PROGRAM MAIN
VAR
END_VAR

Control_FBD();

END_PROGRAM

(* stored: Version 1.1.0.1, ProductVersion 3.1.4022.12
   POU MAIN: Id {4c5f8b35-f0df-4a6f-a8f4-070acba281dc}, SpecialFunc None *)
